{attribute addProperty BoxType "AX5206-0000-0200-0200"}
{attribute addProperty Id "AT_xAT %I*ARRAY[0..1] OF AT_15FCA3A6160200MDTAT %Q*ARRAY[0..1] OF MDT_C2B17B7F96120WcStateAT %I*WcState_F855686C1620InfoDataAT %I*InfoData_81099714160200"}
{attribute addProperty CRC "1322418018"}
{attribute addProperty SizeInBites "432"}
{attribute addProperty SizeInBytes "54"}
TYPE AX5206_08C80E1B :
STRUCT
	{attribute addProperty Name "AT"}
	AT_x : ARRAY[0..1] OF AT_15FCA3A6;
	{attribute addProperty Name "MDT"}
	MDT : ARRAY[0..1] OF MDT_C2B17B7F;
	{attribute addProperty Name "WcState"}
	WcState : WcState_F855686C;
	{attribute addProperty Name "InfoData"}
	InfoData : InfoData_81099714;
END_STRUCT
END_TYPE

(* stored: Version 1.2.0.0, ProductVersion 3.1.4024.9
   DUT AX5206_08C80E1B: Id {2deb5857-dc88-4a94-917b-1cee04e6a27a} *)
